PROGRAM Alarm_Error
VAR
//System_Bit
	Always_ON				:	BOOL	:=TRUE	;//상시 ON
	Always_OFF				:	BOOL	:=FALSE	;//상시 OFF
	Alarm_delay: TON;
END_VAR

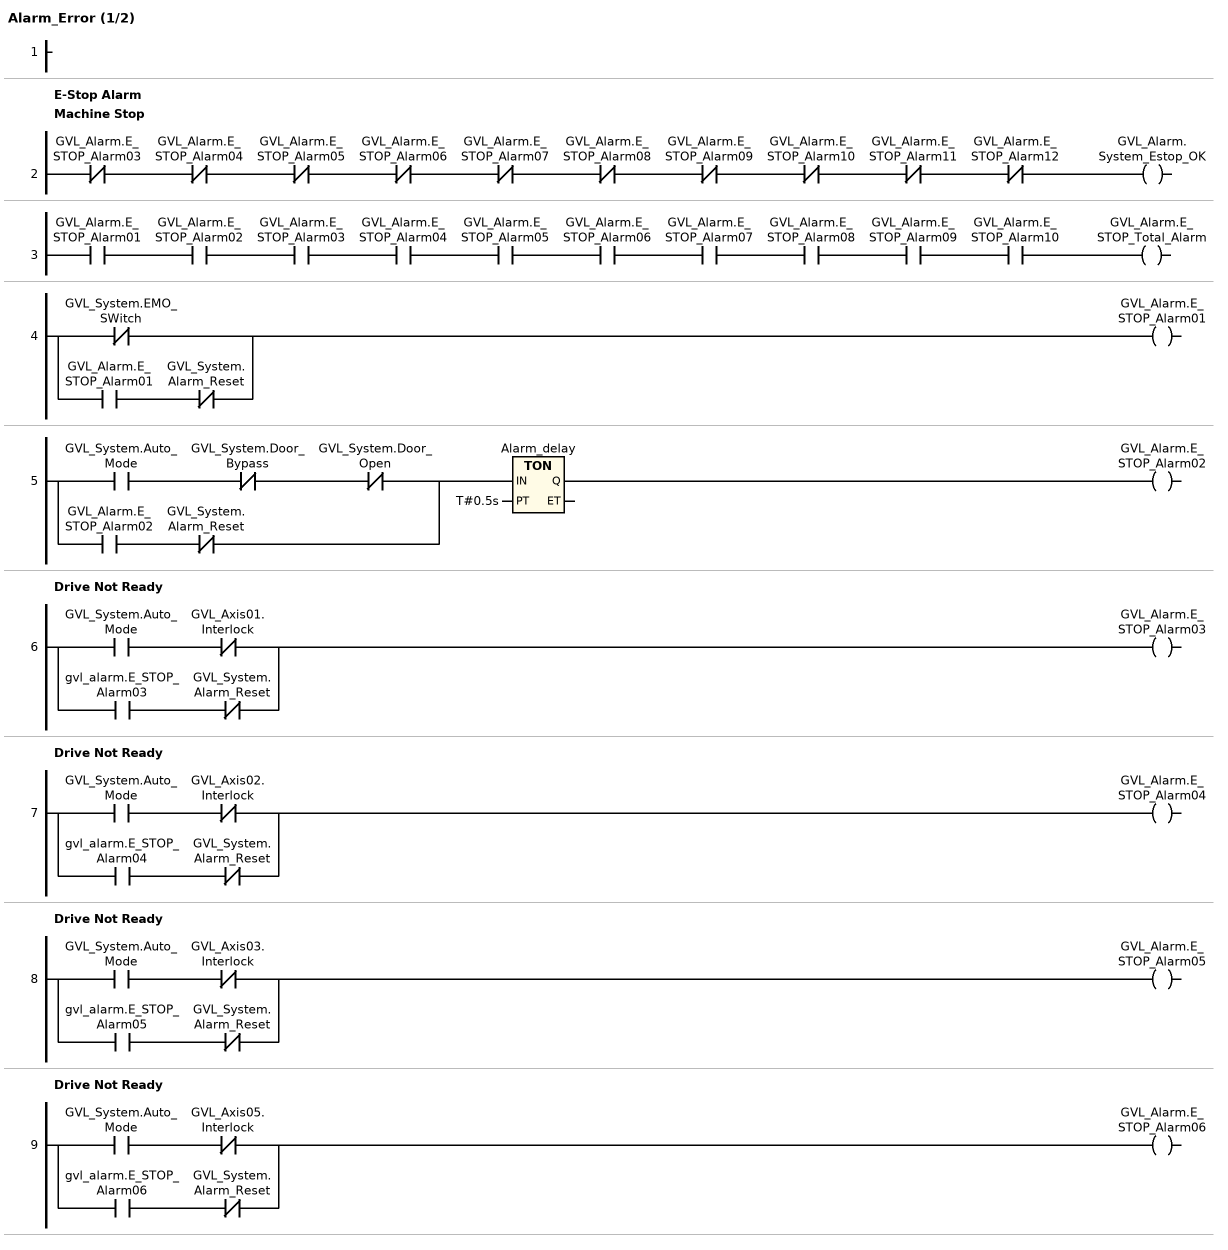
// NETWORK 1

// NETWORK 2: E-Stop Alarm Machine Stop
GVL_Alarm.System_Estop_OK := NOT GVL_Alarm.E_STOP_Alarm03 AND NOT GVL_Alarm.E_STOP_Alarm04 AND NOT GVL_Alarm.E_STOP_Alarm05 AND NOT GVL_Alarm.E_STOP_Alarm06 AND NOT GVL_Alarm.E_STOP_Alarm07 AND NOT GVL_Alarm.E_STOP_Alarm08 AND NOT GVL_Alarm.E_STOP_Alarm09 AND NOT GVL_Alarm.E_STOP_Alarm10 AND NOT GVL_Alarm.E_STOP_Alarm11 AND NOT GVL_Alarm.E_STOP_Alarm12;

// NETWORK 3
GVL_Alarm.E_STOP_Total_Alarm := GVL_Alarm.E_STOP_Alarm01 AND GVL_Alarm.E_STOP_Alarm02 AND GVL_Alarm.E_STOP_Alarm03 AND GVL_Alarm.E_STOP_Alarm04 AND GVL_Alarm.E_STOP_Alarm05 AND GVL_Alarm.E_STOP_Alarm06 AND GVL_Alarm.E_STOP_Alarm07 AND GVL_Alarm.E_STOP_Alarm08 AND GVL_Alarm.E_STOP_Alarm09 AND GVL_Alarm.E_STOP_Alarm10;

// NETWORK 4
GVL_Alarm.E_STOP_Alarm01 := NOT GVL_System.EMO_SWitch OR GVL_Alarm.E_STOP_Alarm01 AND NOT GVL_System.Alarm_Reset;

// NETWORK 5
Alarm_delay(IN := GVL_System.Auto_Mode AND NOT GVL_System.Door_Bypass AND NOT GVL_System.Door_Open OR GVL_Alarm.E_STOP_Alarm02 AND NOT GVL_System.Alarm_Reset, PT := T#0.5s); // TON
GVL_Alarm.E_STOP_Alarm02 := Alarm_delay.Q;

// NETWORK 6: Drive Not Ready
GVL_Alarm.E_STOP_Alarm03 := GVL_System.Auto_Mode AND NOT GVL_Axis01.Interlock OR gvl_alarm.E_STOP_Alarm03 AND NOT GVL_System.Alarm_Reset;

// NETWORK 7: Drive Not Ready
GVL_Alarm.E_STOP_Alarm04 := GVL_System.Auto_Mode AND NOT GVL_Axis02.Interlock OR gvl_alarm.E_STOP_Alarm04 AND NOT GVL_System.Alarm_Reset;

// NETWORK 8: Drive Not Ready
GVL_Alarm.E_STOP_Alarm05 := GVL_System.Auto_Mode AND NOT GVL_Axis03.Interlock OR gvl_alarm.E_STOP_Alarm05 AND NOT GVL_System.Alarm_Reset;

// NETWORK 9: Drive Not Ready
GVL_Alarm.E_STOP_Alarm06 := GVL_System.Auto_Mode AND NOT GVL_Axis05.Interlock OR gvl_alarm.E_STOP_Alarm06 AND NOT GVL_System.Alarm_Reset;

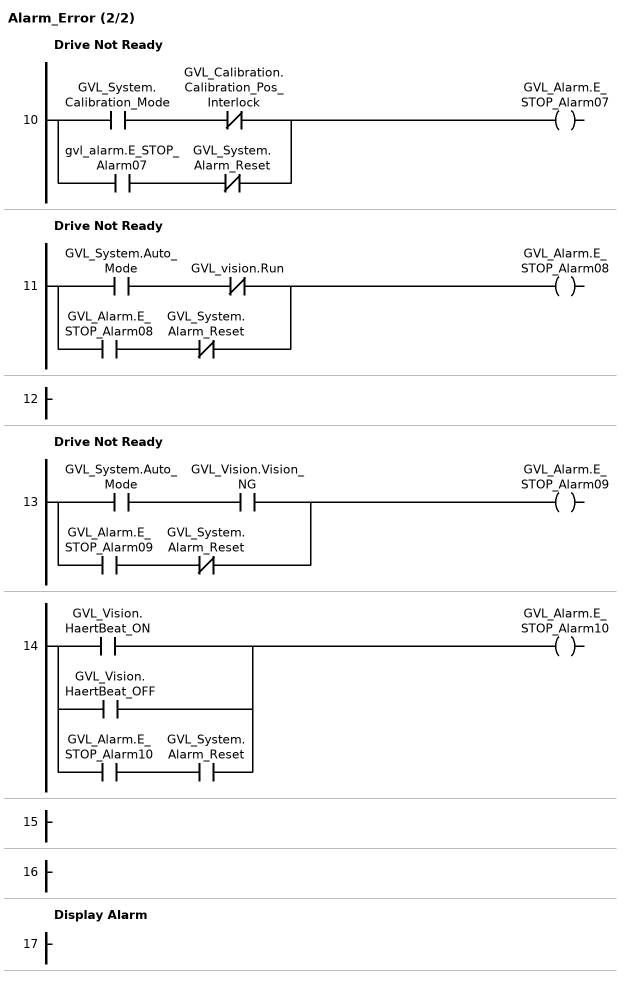
// NETWORK 10: Drive Not Ready
GVL_Alarm.E_STOP_Alarm07 := GVL_System.Calibration_Mode AND NOT GVL_Calibration.Calibration_Pos_Interlock OR gvl_alarm.E_STOP_Alarm07 AND NOT GVL_System.Alarm_Reset;

// NETWORK 11: Drive Not Ready
GVL_Alarm.E_STOP_Alarm08 := GVL_System.Auto_Mode AND NOT GVL_vision.Run OR GVL_Alarm.E_STOP_Alarm08 AND NOT GVL_System.Alarm_Reset;

// NETWORK 12

// NETWORK 13: Drive Not Ready
GVL_Alarm.E_STOP_Alarm09 := GVL_System.Auto_Mode AND GVL_Vision.Vision_NG OR GVL_Alarm.E_STOP_Alarm09 AND NOT GVL_System.Alarm_Reset;

// NETWORK 14
GVL_Alarm.E_STOP_Alarm10 := GVL_Vision.HaertBeat_ON OR GVL_Vision.HaertBeat_OFF OR GVL_Alarm.E_STOP_Alarm10 AND GVL_System.Alarm_Reset;

// NETWORK 15

// NETWORK 16

// NETWORK 17: Display Alarm

END_PROGRAM

(* stored: Version 1.1.0.1, ProductVersion 3.1.4024.15
   POU Alarm_Error: Id {3571cb56-96d6-492b-8474-50953eb81009}, SpecialFunc None *)
